FUNCTION F_CloseDialog : BOOL
VAR_INPUT
	sDialogName : STRING;
END_VAR
VAR
	pstClientData : POINTER TO VisuElems.VisuStructClientData;
	itfDialogManager : VisuElems.IDialogManager;
	itfMyDialog : VisuElems.IVisualisationDialog;
	stVisuRect : VisuElems.VisuStructSimpleRectangle;
END_VAR

VisuElems.VisuElemBase.g_ClientManager.BeginIteration();
pstClientData := VisuElems.VisuElemBase.g_ClientManager.GetNextClient();
WHILE pstClientData <> 0 DO
   IF pstClientData^.GlobalData.ClientType = VisuElems.Visu_ClientType.HMITargetVisualization THEN
      itfDialogManager := VisuElems.g_VisuManager.GetDialogManager();
      itfMyDialog := itfDialogManager.GetDialog(sDialogName);
      itfDialogManager.CloseDialog	(itfMyDialog, pstClientData);
   END_IF
   pstClientData := VisuElems.VisuElemBase.g_ClientManager.GetNextClient();
END_WHILE

END_FUNCTION

(* stored: Version 1.1.0.1, ProductVersion 3.1.4024.9
   POU F_CloseDialog: Id {091be54b-6b74-43eb-8ce6-a17147c37a6b}, SpecialFunc None *)
